(* IEC 61131-3 sources: plc-home-automation/home_automation/lighting_heating_updated/src/utils/slowavg, 1 file *)

(* ---- SlowAvg.st ---- *)
PROGRAM SlowAveraging
  VAR_INPUT
  END_VAR
  VAR_OUTPUT
  END_VAR
  VAR
    window_width : REAL := 150;
  END_VAR
  VAR_TEMP
  END_VAR

  EXTERNAL_AVERAGE_TEMPERATURE := (EXTERNAL_AVERAGE_TEMPERATURE * (window_width - 1) + EXTERNAL_TEMPERATURE) / window_width;

END_PROGRAM
